PROGRAM main
  VAR
    COUNTER1 AT %QW0 : INT;
    STATUS_BIT AT %QX0.0 : BOOL;
    TICK : BOOL;
    T_OFF_DONE : BOOL;
    T_1S : TON;
    C1 : CTU;
    T_ON : TON;
    T_OFF : TON;
    CTU0 : CTU;
    TON0 : TON;
    TON1 : TON;
  END_VAR

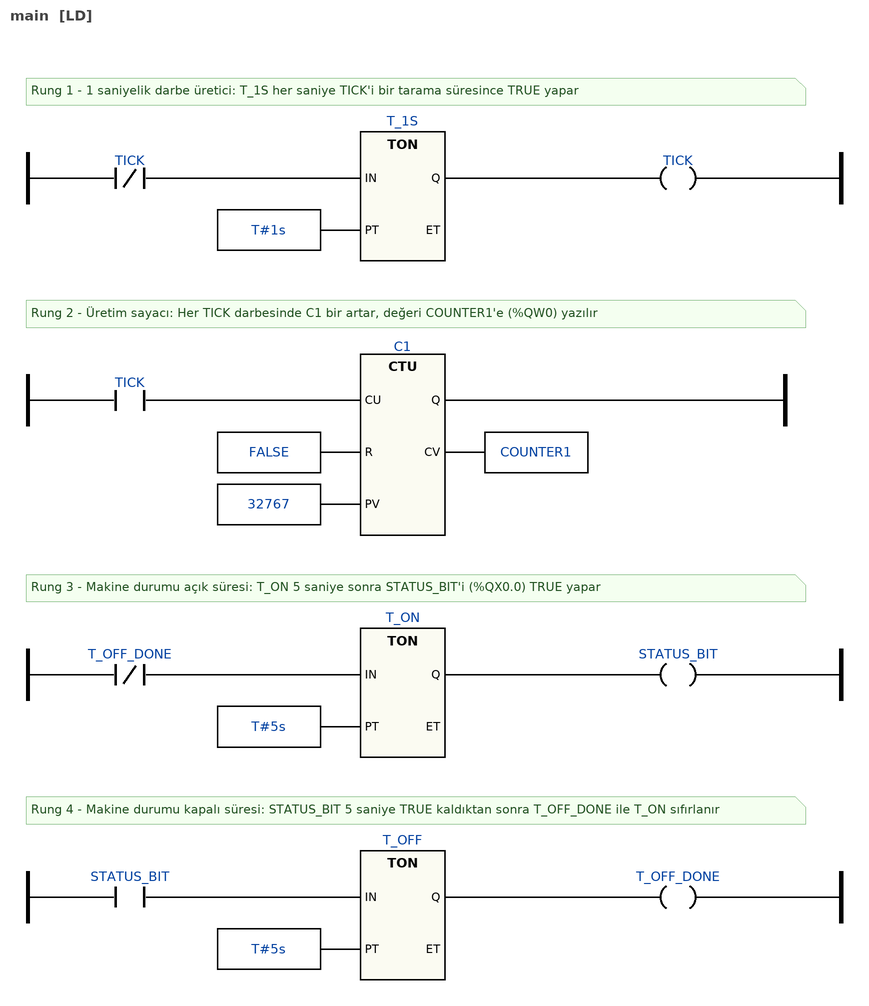
(* LD diagram, written out as Structured Text *)
(* Rung 1 - 1 saniyelik darbe üretici: T_1S her saniye TICK'i bir tarama süresince TRUE yapar *)
T_1S(IN := NOT TICK, PT := T#1s);
TICK := T_1S.Q;
(* Rung 2 - Üretim sayacı: Her TICK darbesinde C1 bir artar, değeri COUNTER1'e (%QW0) yazılır *)
C1(CU := TICK, R := FALSE, PV := 32767);
COUNTER1 := C1.CV;
(* Rung 3 - Makine durumu açık süresi: T_ON 5 saniye sonra STATUS_BIT'i (%QX0.0) TRUE yapar *)
T_ON(IN := NOT T_OFF_DONE, PT := T#5s);
STATUS_BIT := T_ON.Q;
(* Rung 4 - Makine durumu kapalı süresi: STATUS_BIT 5 saniye TRUE kaldıktan sonra T_OFF_DONE ile T_ON sıfırlanır *)
T_OFF(IN := STATUS_BIT, PT := T#5s);
T_OFF_DONE := T_OFF.Q;
END_PROGRAM
